Fanuc KAREL source: kt00910.KL

-- PROVISIONAL review KL for V940-1; original PC SHA256 feecbffee3228d0ab8f8a7de092f43cadaf3479e765fe93bbee9d3ba02e77218
-- Incomplete behavior may be omitted. Consult companion uncertainty JSON. Do not deploy.
PROGRAM KT00910
%NOLOCKGROUP
BEGIN
  -- V9_ZERO_TABLE_METADATA_HINT layout=0002_ascii; no indexed target words; source/name/runtime held
  -- UNRESOLVED_PC offsets 5-20; opcodes 2E,22,32,35
  -- UNRESOLVED_PC offsets 25-40; opcodes 2E,22,32,35
  -- UNRESOLVED_PC offsets 45-60; opcodes 2E,22,32,35
  -- UNRESOLVED_PC offsets 65-80; opcodes 2E,22,32,35
  -- UNRESOLVED_PC offsets 85-111; opcodes 27,27,49,7E,AD,31,4A
  -- UNRESOLVED_PC offsets 116-120; opcodes 7F
END KT00910
